Staubli VAL3: _HomeWatchDog.pgx

public program _HomeWatchDog()
begin
  if taskStatus("resetProgram")!=-1
    //过滤硬件波动
    //    if watch(cycleStatus:bIsHome==true,0)
    if watch(dInGohome==true,0)
    else
      stopMove()
      taskKill("resetProgram")
      watch(taskStatus("resetProgram")==-1,1)
      resetMotion()
    endIf
    if taskStatus("resetProgram")>1
      if taskStatus("resetProgram")>=150 and taskStatus("resetProgram")<=154
        popUpMsg("运动无法到达，超限")
      else
        logMsg("[KERNEL] SUPERVISOR:Task resetProgram problem")
        call OnEvent:OnCycleEvent(12)
      endIf
      stopMove()
      taskKill("resetProgram")
      watch(taskStatus("resetProgram")==-1,1)
      resetMotion()
    endIf
  endIf
end
